(* Logix 5000 project; controller Transcat_L33ER vendor 1 type 14 code 107 rev 32.11; software revision 32.02; part 2 of 4 *)
(* tags used below, declared in another part *)
   AcsiiToReal1 : HexASCII_to_REAL;
   AnyAutoRun : BOOL;   // Bit that in on if ANY device is placed into Auto run (to signal pre-start beed)
   AnyAutoRunFlag : BOOL;   // A flag that indicates if any device is in Auto Run (used with pre-start beep logic)
   AnyManRunFlag : BOOL;   // A flag that indicates if any device is in Manual Run (used with pre-start beep logic)
   AnyManualRun : BOOL;   // Bit that in on if ANY device is placed into manual run (to signal pre-start beed)
   AutoActive : BOOL;   // Auto mode active
   AutoStartOS : BOOL;   // Auto Start One-Shot
   AutoStopOS : BOOL;   // Auto Stop One-Shot
   Beep : BOOL;   // Bit to Activte Beacon Alarm
   bronkhorstReal : REAL[50];   // data from Bonkhorst - convertred to real values
   BronkOutArr : DINT[3];   // 3 Outputs from Flow controllers 0 - 100% = 0 - 32000
   BronkRealInArr : REAL[100];
   ConversionError : BOOL;
   ConvertedFloat : REAL;
   CV_101_Output : ALIAS FOR TC_Remote_IO:5:O.1;   // CV_101 - 3 Way Valve - Recyle / Process
   dataIndex : DINT;   // Bronkhorst Data Index
   Device : Device[20];
   FT103 : BronkhorstFlowMeter;
   FT103B : BronkhorstFlowMeter;
   FT104 : BronkhorstFlowMeter;
   FT104B : BronkhorstFlowMeter;
   FT105 : BronkhorstFlowMeter;
   FT105B : BronkhorstFlowMeter;
   HMI_AutoStart : BOOL;   // Starts all devices in AUTO
   HMI_AutoStop : BOOL;   // Stops all devices in AUTO
   MX101 : Howes_Mixer;
   NewDataToggle : BOOL;
   PT103_PV_RAW : ALIAS FOR TC_Remote_IO:1:I.Ch0Data;   // Raw (unscaled) pressure reading from PT103 - PSI * 100 (range 0 - 108 PSI)
   PT104_PV_RAW : ALIAS FOR TC_Remote_IO:1:I.Ch1Data;   // Raw (unscaled) pressure reading from PT104 - PSI * 100 (range 0 - 108 PSI)
   PT105_PV_RAW : ALIAS FOR TC_Remote_IO:1:I.Ch2Data;   // Raw (unscaled) pressure reading from PT105 - PSI * 100 (range 0 - 108 PSI)
   resultIndex : DINT;   // Bronkhorst Real Result Index
   SC1 : Howes_Mixer;   // UDT for screener
   TempHexIn : SINT[8];   // Place to copy 8 SINT for proessing by AOI
   VF201 : Acrison_Feeder;   // Small Feeder 2 Tags
(* MainProgram, continued *)

ROUTINE _06_VF201_Small_Feeder_2   (* ladder *)
// Acison Small Feeder Control
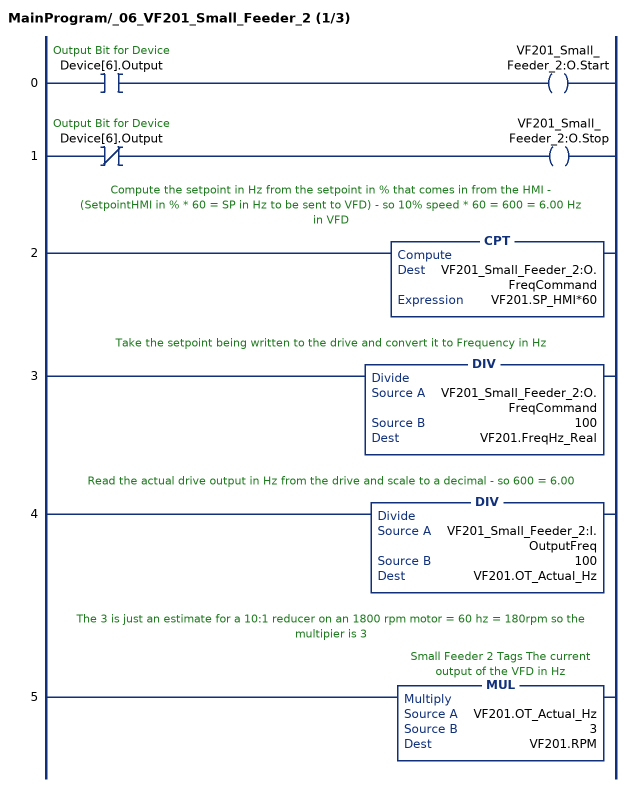
   0: XIC(Device[6].Output)OTE(VF201_Small_Feeder_2:O.Start);
   1: XIO(Device[6].Output)OTE(VF201_Small_Feeder_2:O.Stop);
   // Compute the setpoint in Hz from the setpoint in % that comes in from the HMI - (SetpointHMI in % * 60 = SP in Hz to be sent to VFD) - so 10% speed * 60 = 600 = 6.00 Hz in VFD
   2: CPT(VF201_Small_Feeder_2:O.FreqCommand,VF201.SP_HMI*60);
   // Take the setpoint being written to the drive and convert it to Frequency in Hz
   3: DIV(VF201_Small_Feeder_2:O.FreqCommand,100,VF201.FreqHz_Real);
   // Read the actual drive output in Hz from the drive and scale to a decimal - so 600 = 6.00
   4: DIV(VF201_Small_Feeder_2:I.OutputFreq,100,VF201.OT_Actual_Hz);
   // The 3 is just an estimate for a 10:1 reducer on an 1800 rpm motor = 60 hz = 180rpm so the multipier is 3
   5: MUL(VF201.OT_Actual_Hz,3,VF201.RPM);
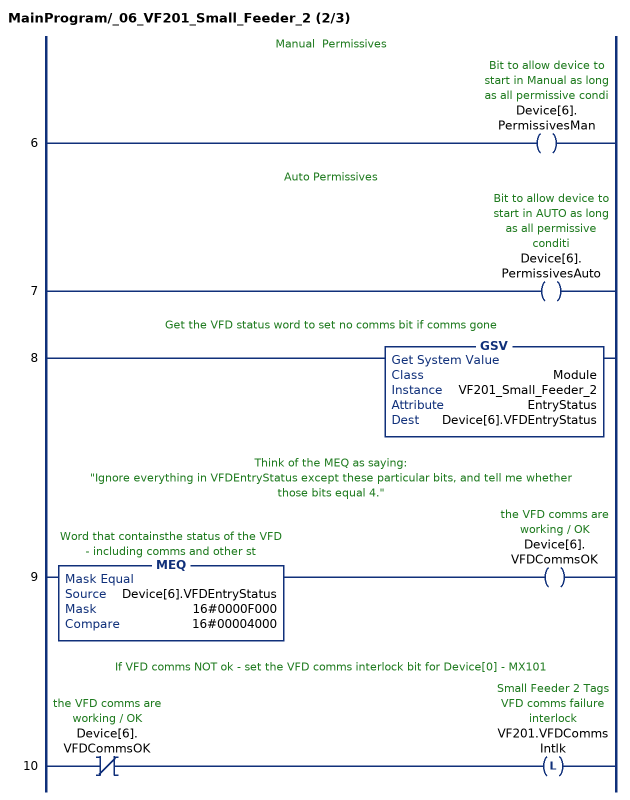
   // Manual  Permissives
   6: OTE(Device[6].PermissivesMan);
   // Auto Permissives
   7: OTE(Device[6].PermissivesAuto);
   // Get the VFD status word to set no comms bit if comms gone
   8: GSV(Module,VF201_Small_Feeder_2,EntryStatus,Device[6].VFDEntryStatus);
   // Think of the MEQ as saying:
   // "Ignore everything in VFDEntryStatus except these particular bits, and tell me whether those bits equal 4."
   9: MEQ(Device[6].VFDEntryStatus,16#0000F000,16#00004000)OTE(Device[6].VFDCommsOK);
   // If VFD comms NOT ok - set the VFD comms interlock bit for Device[0] - MX101
   10: XIO(Device[6].VFDCommsOK)OTL(VF201.VFDCommsIntlk);
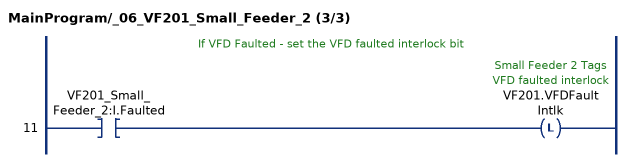
   // If VFD Faulted - set the VFD faulted interlock bit
   11: XIC(VF201_Small_Feeder_2:I.Faulted)OTL(VF201.VFDFaultIntlk);
END_ROUTINE

ROUTINE _07_FT103_Oil_Dosing   (* ladder *)
// Logic to control FT103 not associated with Device Iteration Logic
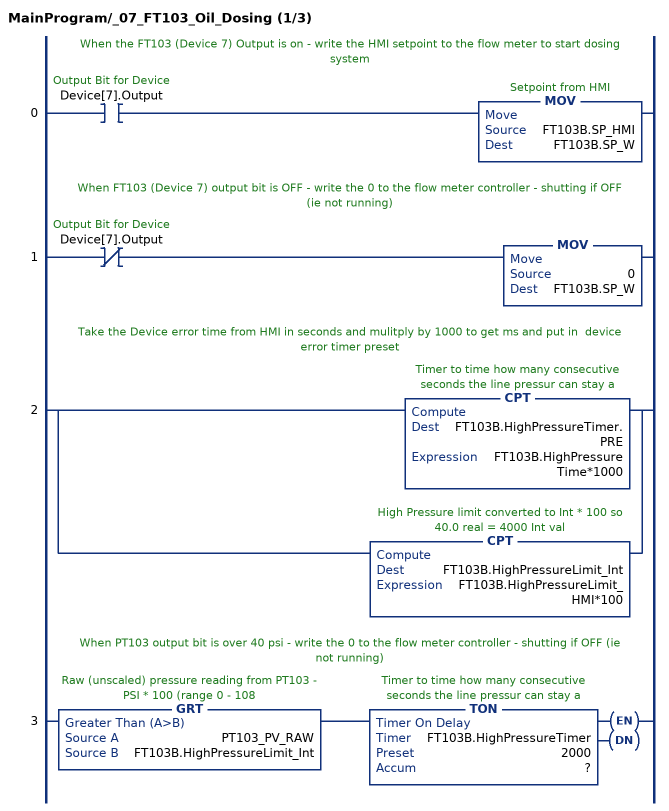
   // When the FT103 (Device 7) Output is on - write the HMI setpoint to the flow meter to start dosing system
   0: XIC(Device[7].Output)MOV(FT103B.SP_HMI,FT103B.SP_W);
   // When FT103 (Device 7) output bit is OFF - write the 0 to the flow meter controller - shutting if OFF (ie not running)
   1: XIO(Device[7].Output)MOV(0,FT103B.SP_W);
   // Take the Device error time from HMI in seconds and mulitply by 1000 to get ms and put in  device error timer preset
   2: [CPT(FT103B.HighPressureTimer.PRE,FT103B.HighPressureTime*1000) ,CPT(FT103B.HighPressureLimit_Int,FT103B.HighPressureLimit_HMI*100) ];
   // When PT103 output bit is over 40 psi - write the 0 to the flow meter controller - shutting if OFF (ie not running)
   3: GRT(PT103_PV_RAW,FT103B.HighPressureLimit_Int)TON(FT103B.HighPressureTimer,?,?);
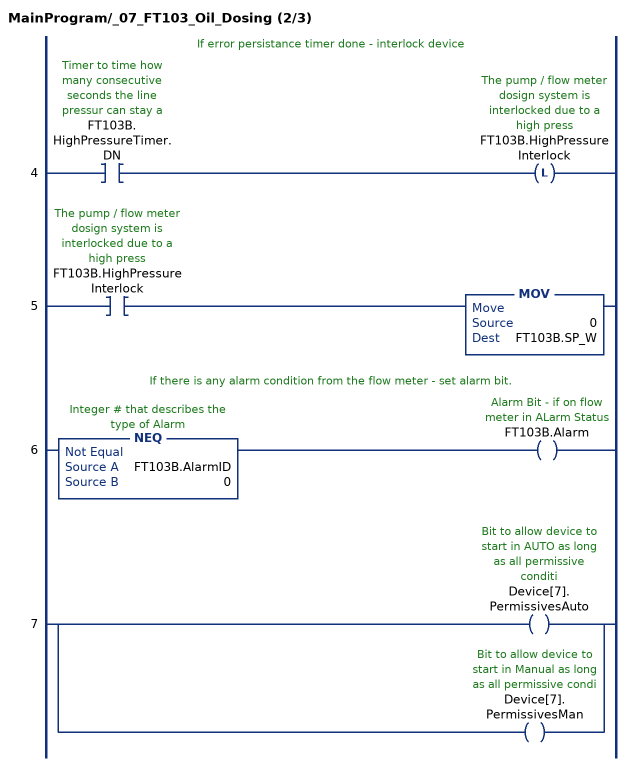
   // If error persistance timer done - interlock device
   4: XIC(FT103B.HighPressureTimer.DN)OTL(FT103B.HighPressureInterlock);
   5: XIC(FT103B.HighPressureInterlock)MOV(0,FT103B.SP_W);
   // If there is any alarm condition from the flow meter - set alarm bit.
   6: NEQ(FT103B.AlarmID,0)OTE(FT103B.Alarm);
   7: [OTE(Device[7].PermissivesAuto) ,OTE(Device[7].PermissivesMan) ];
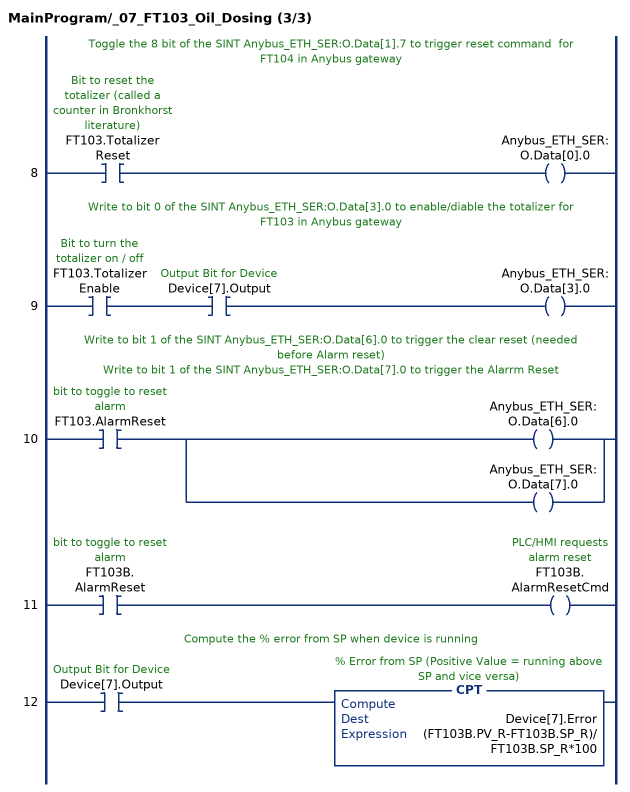
   // Toggle the 8 bit of the SINT Anybus_ETH_SER:O.Data[1].7 to trigger reset command  for FT104 in Anybus gateway
   8: XIC(FT103.TotalizerReset)OTE(Anybus_ETH_SER:O.Data[0].0);
   // Write to bit 0 of the SINT Anybus_ETH_SER:O.Data[3].0 to enable/diable the totalizer for FT103 in Anybus gateway
   9: XIC(FT103.TotalizerEnable)XIC(Device[7].Output)OTE(Anybus_ETH_SER:O.Data[3].0);
   // Write to bit 1 of the SINT Anybus_ETH_SER:O.Data[6].0 to trigger the clear reset (needed before Alarm reset)
   // Write to bit 1 of the SINT Anybus_ETH_SER:O.Data[7].0 to trigger the Alarrm Reset
   10: XIC(FT103.AlarmReset)[OTE(Anybus_ETH_SER:O.Data[6].0) ,OTE(Anybus_ETH_SER:O.Data[7].0) ];
   11: XIC(FT103B.AlarmReset)OTE(FT103B.AlarmResetCmd);
   // Compute the % error from SP when device is running
   12: XIC(Device[7].Output)CPT(Device[7].Error,(FT103B.PV_R-FT103B.SP_R)/FT103B.SP_R*100);
END_ROUTINE

ROUTINE _08_FT104_Water_Dosing   (* ladder *)
// FT104 Control Logic not associated with Device Iteration Logic
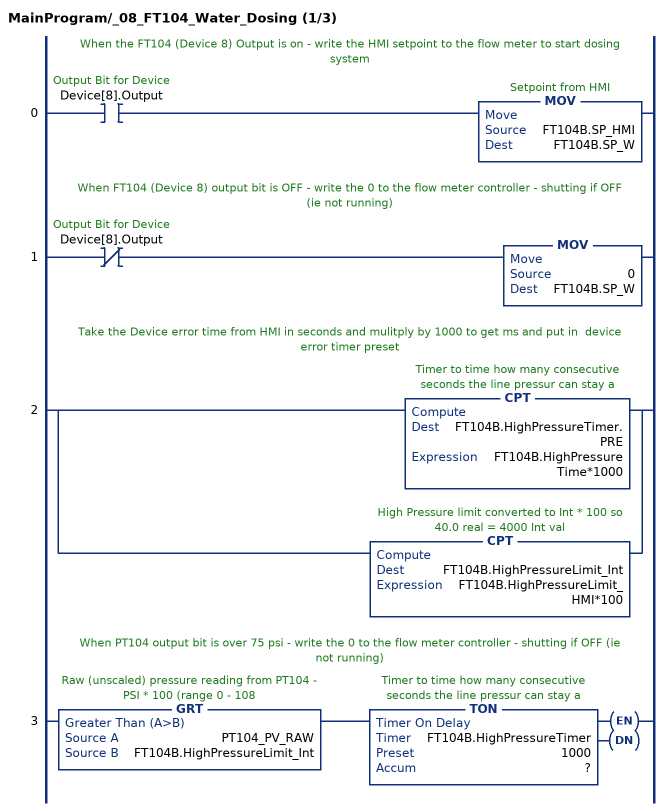
   // When the FT104 (Device 8) Output is on - write the HMI setpoint to the flow meter to start dosing system
   0: XIC(Device[8].Output)MOV(FT104B.SP_HMI,FT104B.SP_W);
   // When FT104 (Device 8) output bit is OFF - write the 0 to the flow meter controller - shutting if OFF (ie not running)
   1: XIO(Device[8].Output)MOV(0,FT104B.SP_W);
   // Take the Device error time from HMI in seconds and mulitply by 1000 to get ms and put in  device error timer preset
   2: [CPT(FT104B.HighPressureTimer.PRE,FT104B.HighPressureTime*1000) ,CPT(FT104B.HighPressureLimit_Int,FT104B.HighPressureLimit_HMI*100) ];
   // When PT104 output bit is over 75 psi - write the 0 to the flow meter controller - shutting if OFF (ie not running)
   3: GRT(PT104_PV_RAW,FT104B.HighPressureLimit_Int)TON(FT104B.HighPressureTimer,?,?);
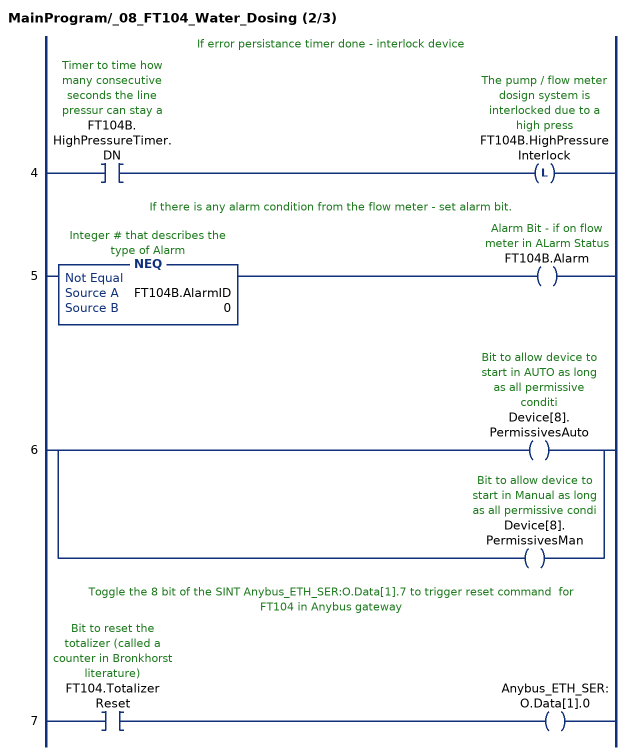
   // If error persistance timer done - interlock device
   4: XIC(FT104B.HighPressureTimer.DN)OTL(FT104B.HighPressureInterlock);
   // If there is any alarm condition from the flow meter - set alarm bit.
   5: NEQ(FT104B.AlarmID,0)OTE(FT104B.Alarm);
   6: [OTE(Device[8].PermissivesAuto) ,OTE(Device[8].PermissivesMan) ];
   // Toggle the 8 bit of the SINT Anybus_ETH_SER:O.Data[1].7 to trigger reset command  for FT104 in Anybus gateway
   7: XIC(FT104.TotalizerReset)OTE(Anybus_ETH_SER:O.Data[1].0);
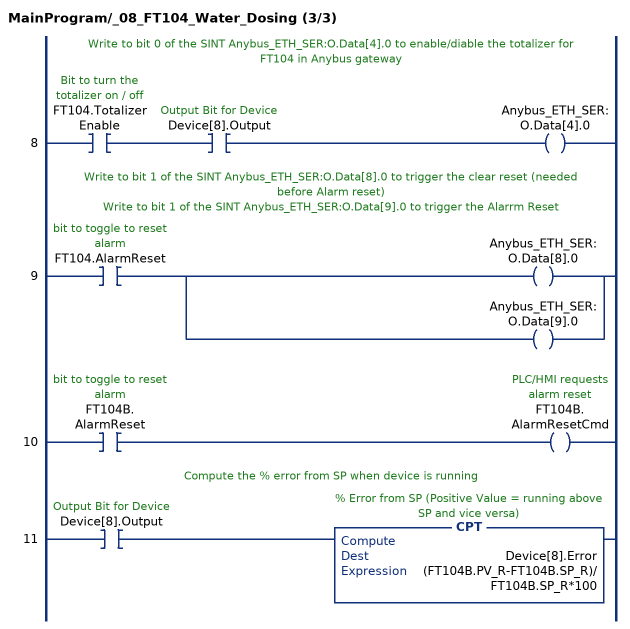
   // Write to bit 0 of the SINT Anybus_ETH_SER:O.Data[4].0 to enable/diable the totalizer for FT104 in Anybus gateway
   8: XIC(FT104.TotalizerEnable)XIC(Device[8].Output)OTE(Anybus_ETH_SER:O.Data[4].0);
   // Write to bit 1 of the SINT Anybus_ETH_SER:O.Data[8].0 to trigger the clear reset (needed before Alarm reset)
   // Write to bit 1 of the SINT Anybus_ETH_SER:O.Data[9].0 to trigger the Alarrm Reset
   9: XIC(FT104.AlarmReset)[OTE(Anybus_ETH_SER:O.Data[8].0) ,OTE(Anybus_ETH_SER:O.Data[9].0) ];
   10: XIC(FT104B.AlarmReset)OTE(FT104B.AlarmResetCmd);
   // Compute the % error from SP when device is running
   11: XIC(Device[8].Output)CPT(Device[8].Error,(FT104B.PV_R-FT104B.SP_R)/FT104B.SP_R*100);
END_ROUTINE

ROUTINE _09_FT105_Fragrance_Dosing   (* ladder *)
// FT105 Control Logic not associated with Device Iteration Logic
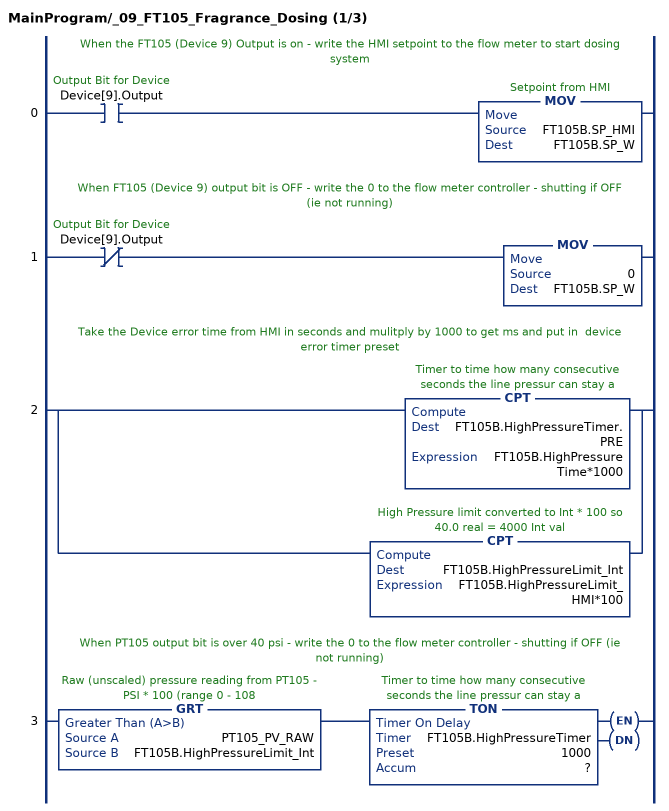
   // When the FT105 (Device 9) Output is on - write the HMI setpoint to the flow meter to start dosing system
   0: XIC(Device[9].Output)MOV(FT105B.SP_HMI,FT105B.SP_W);
   // When FT105 (Device 9) output bit is OFF - write the 0 to the flow meter controller - shutting if OFF (ie not running)
   1: XIO(Device[9].Output)MOV(0,FT105B.SP_W);
   // Take the Device error time from HMI in seconds and mulitply by 1000 to get ms and put in  device error timer preset
   2: [CPT(FT105B.HighPressureTimer.PRE,FT105B.HighPressureTime*1000) ,CPT(FT105B.HighPressureLimit_Int,FT105B.HighPressureLimit_HMI*100) ];
   // When PT105 output bit is over 40 psi - write the 0 to the flow meter controller - shutting if OFF (ie not running)
   3: GRT(PT105_PV_RAW,FT105B.HighPressureLimit_Int)TON(FT105B.HighPressureTimer,?,?);
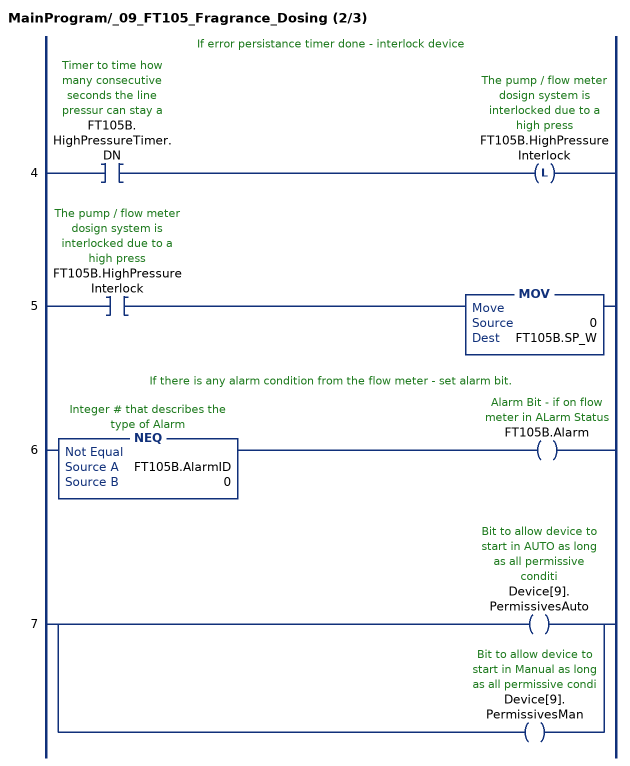
   // If error persistance timer done - interlock device
   4: XIC(FT105B.HighPressureTimer.DN)OTL(FT105B.HighPressureInterlock);
   5: XIC(FT105B.HighPressureInterlock)MOV(0,FT105B.SP_W);
   // If there is any alarm condition from the flow meter - set alarm bit.
   6: NEQ(FT105B.AlarmID,0)OTE(FT105B.Alarm);
   7: [OTE(Device[9].PermissivesAuto) ,OTE(Device[9].PermissivesMan) ];
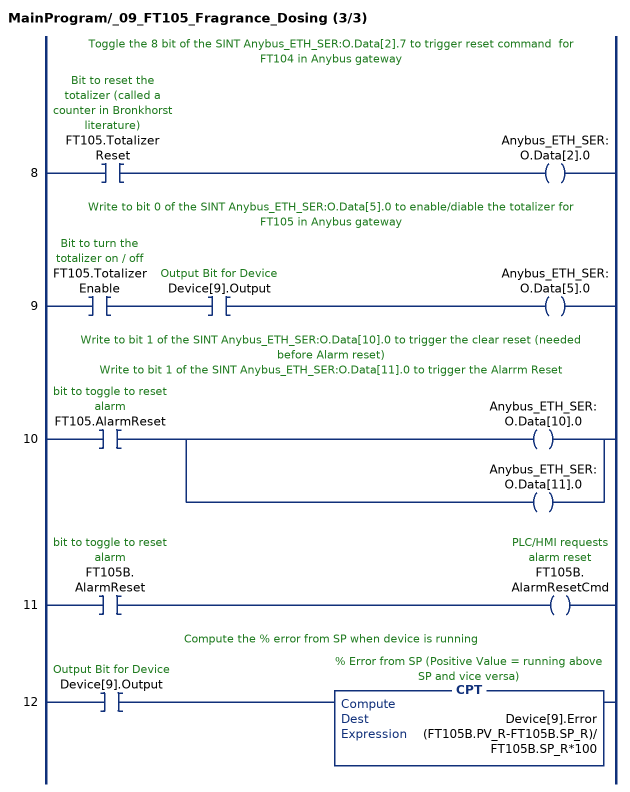
   // Toggle the 8 bit of the SINT Anybus_ETH_SER:O.Data[2].7 to trigger reset command  for FT104 in Anybus gateway
   8: XIC(FT105.TotalizerReset)OTE(Anybus_ETH_SER:O.Data[2].0);
   // Write to bit 0 of the SINT Anybus_ETH_SER:O.Data[5].0 to enable/diable the totalizer for FT105 in Anybus gateway
   9: XIC(FT105.TotalizerEnable)XIC(Device[9].Output)OTE(Anybus_ETH_SER:O.Data[5].0);
   // Write to bit 1 of the SINT Anybus_ETH_SER:O.Data[10].0 to trigger the clear reset (needed before Alarm reset)
   // Write to bit 1 of the SINT Anybus_ETH_SER:O.Data[11].0 to trigger the Alarrm Reset
   10: XIC(FT105.AlarmReset)[OTE(Anybus_ETH_SER:O.Data[10].0) ,OTE(Anybus_ETH_SER:O.Data[11].0) ];
   11: XIC(FT105B.AlarmReset)OTE(FT105B.AlarmResetCmd);
   // Compute the % error from SP when device is running
   12: XIC(Device[9].Output)CPT(Device[9].Error,(FT105B.PV_R-FT105B.SP_R)/FT105B.SP_R*100);
END_ROUTINE

ROUTINE _11_Auxillary_Pump_AE   (* ladder *)
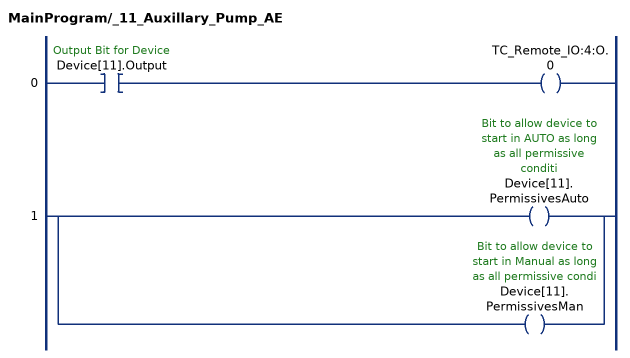
   0: XIC(Device[11].Output)OTE(TC_Remote_IO:4:O.0);
   1: [OTE(Device[11].PermissivesAuto) ,OTE(Device[11].PermissivesMan) ];
END_ROUTINE

ROUTINE _12_SC_1_Screener   (* ladder *)
// Screener
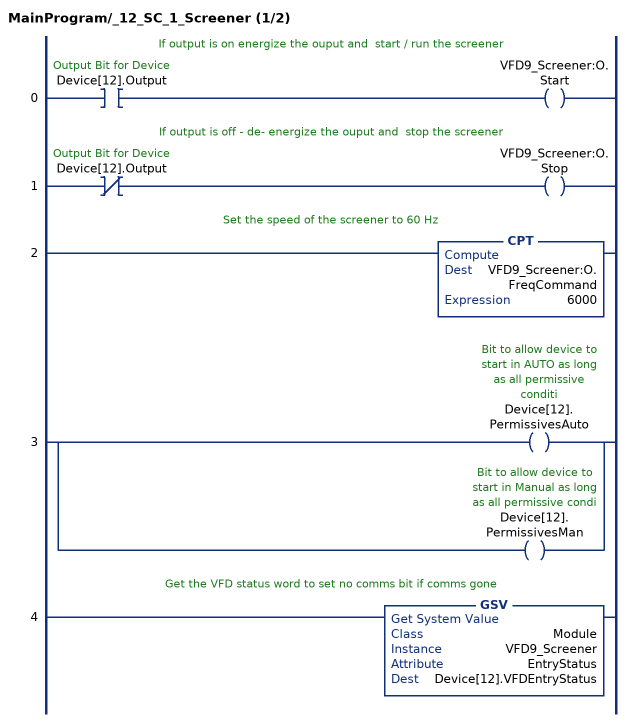
   // If output is on energize the ouput and  start / run the screener
   0: XIC(Device[12].Output)OTE(VFD9_Screener:O.Start);
   // If output is off - de- energize the ouput and  stop the screener
   1: XIO(Device[12].Output)OTE(VFD9_Screener:O.Stop);
   // Set the speed of the screener to 60 Hz
   2: CPT(VFD9_Screener:O.FreqCommand,6000);
   3: [OTE(Device[12].PermissivesAuto) ,OTE(Device[12].PermissivesMan) ];
   // Get the VFD status word to set no comms bit if comms gone
   4: GSV(Module,VFD9_Screener,EntryStatus,Device[12].VFDEntryStatus);
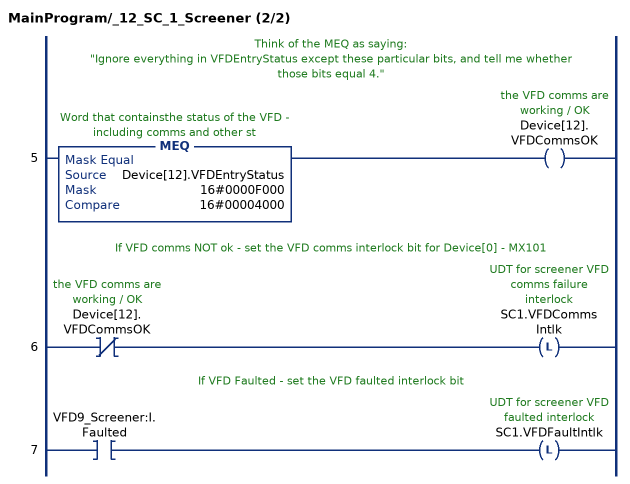
   // Think of the MEQ as saying:
   // "Ignore everything in VFDEntryStatus except these particular bits, and tell me whether those bits equal 4."
   5: MEQ(Device[12].VFDEntryStatus,16#0000F000,16#00004000)OTE(Device[12].VFDCommsOK);
   // If VFD comms NOT ok - set the VFD comms interlock bit for Device[0] - MX101
   6: XIO(Device[12].VFDCommsOK)OTL(SC1.VFDCommsIntlk);
   // If VFD Faulted - set the VFD faulted interlock bit
   7: XIC(VFD9_Screener:I.Faulted)OTL(SC1.VFDFaultIntlk);
END_ROUTINE

ROUTINE _13_CV101_3_Way_Dosing_Value   (* ladder *)
// 3 way valve to switch between recyle and feed to process
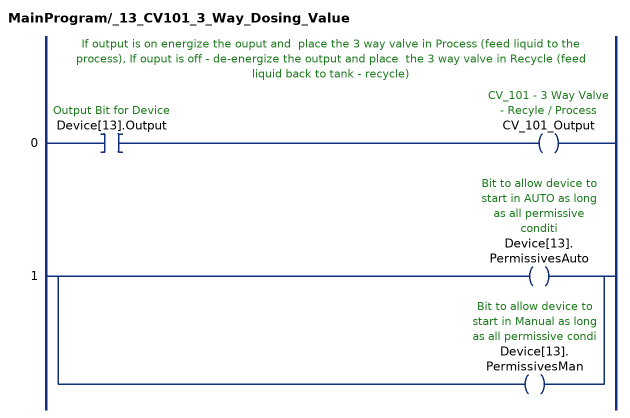
   // If output is on energize the ouput and  place the 3 way valve in Process (feed liquid to the process), If ouput is off - de-energize the output and place  the 3 way valve in Recycle (feed liquid back to tank - recycle)
   0: XIC(Device[13].Output)OTE(CV_101_Output);
   1: [OTE(Device[13].PermissivesAuto) ,OTE(Device[13].PermissivesMan) ];
END_ROUTINE

ROUTINE AutoControl   (* ladder *)
// Place where Auto device control logic lives
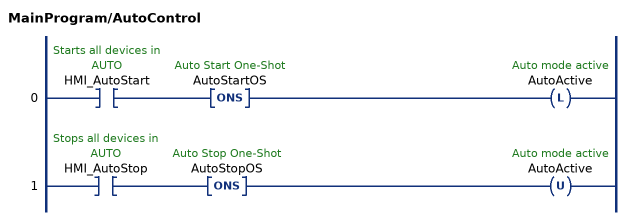
   0: XIC(HMI_AutoStart)ONS(AutoStartOS)OTL(AutoActive);
   1: XIC(HMI_AutoStop)ONS(AutoStopOS)OTU(AutoActive);
END_ROUTINE

ROUTINE BronkDataMapping   (* structured text *)
// Map FT UDT elements to data to/from Bronkhorst Anybus Gateway
   FT103.AlarmID := Anybus_ETH_SER:I.Data[200];
   FT104.AlarmID := Anybus_ETH_SER:I.Data[201];
   FT105.AlarmID := Anybus_ETH_SER:I.Data[202];
   
   FT103.PV_R := BronkRealInArr[0];
   FT103.TempC := BronkRealInArr[1];
   FT103.Density := BronkRealInArr[2];
   FT103.SP_R := BronkRealInArr[3];
   FT103.Totalizer := BronkRealInArr[4];
   
   FT104.PV_R := BronkRealInArr[5];
   FT104.TempC := BronkRealInArr[6];
   FT104.Density := BronkRealInArr[7];
   FT104.SP_R := BronkRealInArr[8];
   FT104.Totalizer := BronkRealInArr[9];
   
   FT105.PV_R := BronkRealInArr[10];
   FT105.TempC := BronkRealInArr[11];
   FT105.Density := BronkRealInArr[12];
   FT105.SP_R := BronkRealInArr[13];
   FT105.Totalizer := BronkRealInArr[14];
   
   FT103.OT_R := (BronkOutArr[0]) / 167681.5;
   FT104.OT_R := (BronkOutArr[1]) / 167681.5;
   FT105.OT_R := (BronkOutArr[2]) / 167681.5;
END_ROUTINE

ROUTINE Bronkhorst_Data   (* ladder *)
// read and write data to/from the EIP instance and convert to/from 8 byte to/from floating point
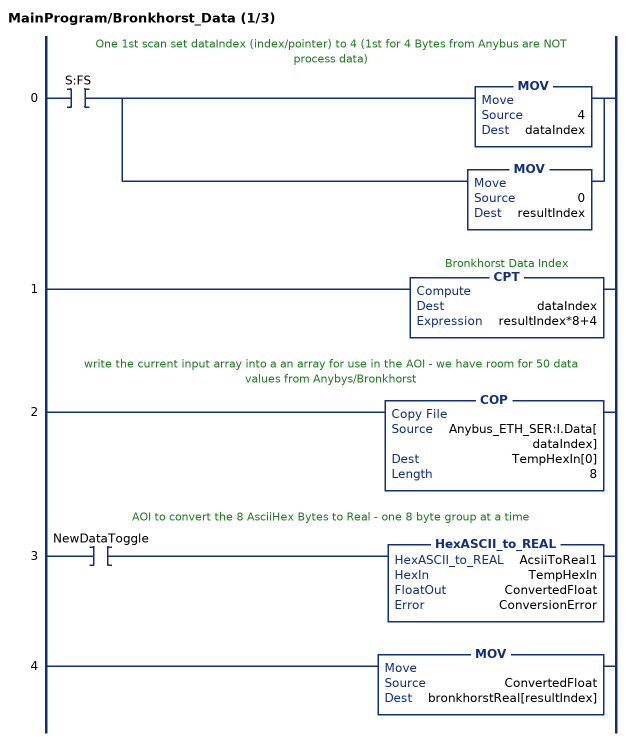
   // One 1st scan set dataIndex (index/pointer) to 4 (1st for 4 Bytes from Anybus are NOT process data)
   0: XIC(S:FS)[MOV(4,dataIndex) ,MOV(0,resultIndex) ];
   1: CPT(dataIndex,resultIndex*8+4);
   // write the current input array into a an array for use in the AOI - we have room for 50 data values from Anybys/Bronkhorst
   2: COP(Anybus_ETH_SER:I.Data[dataIndex],TempHexIn[0],8);
   // AOI to convert the 8 AsciiHex Bytes to Real - one 8 byte group at a time
   3: XIC(NewDataToggle)HexASCII_to_REAL(AcsiiToReal1,TempHexIn,ConvertedFloat,ConversionError);
   4: MOV(ConvertedFloat,bronkhorstReal[resultIndex]);
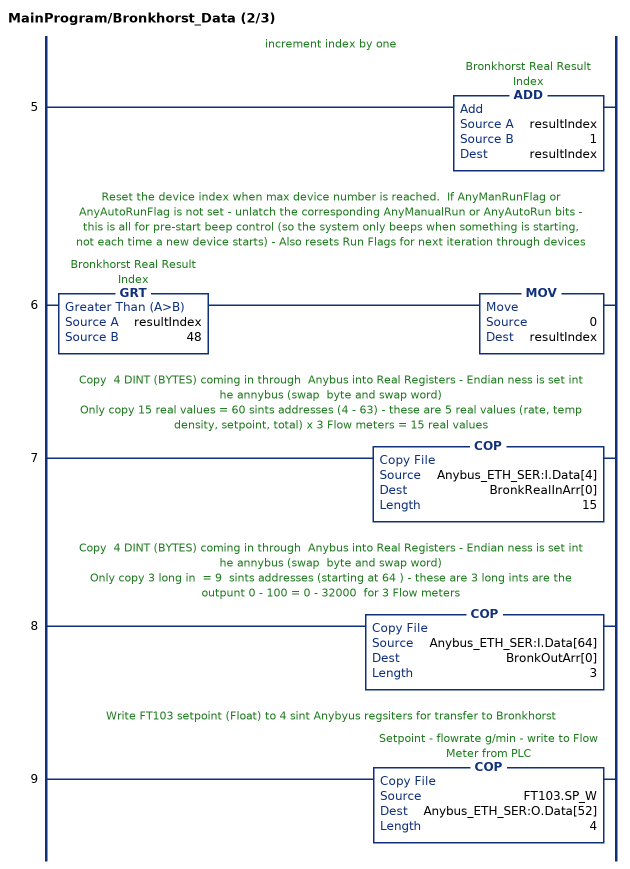
   // increment index by one
   5: ADD(resultIndex,1,resultIndex);
   // Reset the device index when max device number is reached.  If AnyManRunFlag or AnyAutoRunFlag is not set - unlatch the corresponding AnyManualRun or AnyAutoRun bits - this is all for pre-start beep control (so the system only beeps when something is starting, not each time a new device starts) - Also resets Run Flags for next iteration through devices
   6: GRT(resultIndex,48)MOV(0,resultIndex);
   // Copy  4 DINT (BYTES) coming in through  Anybus into Real Registers - Endian ness is set int he annybus (swap  byte and swap word)
   // Only copy 15 real values = 60 sints addresses (4 - 63) - these are 5 real values (rate, temp density, setpoint, total) x 3 Flow meters = 15 real values
   7: COP(Anybus_ETH_SER:I.Data[4],BronkRealInArr[0],15);
   // Copy  4 DINT (BYTES) coming in through  Anybus into Real Registers - Endian ness is set int he annybus (swap  byte and swap word)
   // Only copy 3 long in  = 9  sints addresses (starting at 64 ) - these are 3 long ints are the outpunt 0 - 100 = 0 - 32000  for 3 Flow meters
   8: COP(Anybus_ETH_SER:I.Data[64],BronkOutArr[0],3);
   // Write FT103 setpoint (Float) to 4 sint Anybyus regsiters for transfer to Bronkhorst
   9: COP(FT103.SP_W,Anybus_ETH_SER:O.Data[52],4);
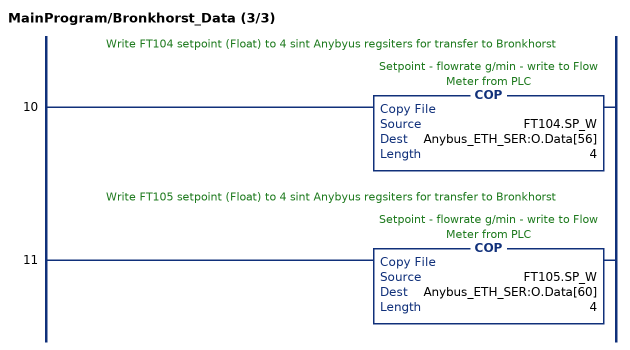
   // Write FT104 setpoint (Float) to 4 sint Anybyus regsiters for transfer to Bronkhorst
   10: COP(FT104.SP_W,Anybus_ETH_SER:O.Data[56],4);
   // Write FT105 setpoint (Float) to 4 sint Anybyus regsiters for transfer to Bronkhorst
   11: COP(FT105.SP_W,Anybus_ETH_SER:O.Data[60],4);
END_ROUTINE
